// Alarm siren FB
FUNCTION_BLOCK FB_AlarmSiren IMPLEMENTS I_AlarmSiren
VAR
	sName				: STRING;				// Siren name
	nID					: INT;					// Alarm component ID
	
	ibTamper			AT %I* : BOOL;			// Active low tamper input
	fbLight				: FB_DigitalOut;		// Siren light digital output FB
	fbSiren				: FB_DigitalOut;		// Siren sound digital output FB
	
	bTamper				: BOOL;					// True if the siren is tampered with
	
	bTamperTrigger		: BOOL;					// True when the tamper sensor is triggered (one cycle)
	
	stHMI				: ST_AlarmSirenHMI;		// HMI data
END_VAR

// Run this method every cycle
METHOD Execute
VAR_INST
	fbTamper	: R_TRIG;		// Tamper rising edge
END_VAR
// Convert active low inputs
bTamper := NOT ibTamper;

// Run FBs
fbTamper(CLK := bTamper);

// Check trigger
bTamperTrigger := fbTamper.Q;

// Update HMI
UpdateHMI();
END_METHOD

METHOD FB_init : BOOL
VAR_INPUT
	bInitRetains	: BOOL;		// if TRUE, the retain variables are initialized (warm start / cold start)
	bInCopyCode		: BOOL;		// if TRUE, the instance afterwards gets moved into the copy code (online change)
	
	sSirenName		: STRING;	// Siren name
	nSirenID		: INT;		// Sensor ID
END_VAR
sName := sSirenName;
nID := nSirenID;
END_METHOD

// Returns the HMI data
PROPERTY HmiData : ST_AlarmSirenHMI
GET
HmiData := stHMI;
END_GET
END_PROPERTY

// Get the alarm component ID of the siren
PROPERTY ID : INT
GET
ID := nID;
END_GET
END_PROPERTY

// Set siren light
METHOD SetLight
VAR_INPUT
	eCommand	: E_DOCommand;		// Siren digital output command
END_VAR
// Set siren digital output command
fbLight.SetCommand(eCommandIn := eCommand);
END_METHOD

// Set siren sound
METHOD SetSound
VAR_INPUT
	eCommand	: E_DOCommand;		// Siren sound digital output command
END_VAR
// Set the siren digital output command
fbSiren.SetCommand(eCommandIn := eCommand);
END_METHOD

// Returns true when the siren is tampered with (as long as the siren is tampered with)
PROPERTY Tamper : BOOL
GET
Tamper := bTamper;
END_GET
END_PROPERTY

// Returns true when the tamper sensor is triggered (one cycle)
PROPERTY TamperTrigger : BOOL
GET
TamperTrigger := bTamperTrigger;
END_GET
END_PROPERTY

// Update HMI
METHOD PRIVATE UpdateHMI
VAR
	stSirenHMI	: ST_HmiDigitalOut;
	stLightHMI	: ST_HmiDigitalOut;
END_VAR
// Get data
stSirenHMI := fbSiren.HmiData;
stLightHMI := fbLight.HmiData;

// Set HMI data
stHMI.sName := sName;
stHMI.nID := nID;
stHMI.bSiren := stSirenHMI.bValue;
stHMI.bLight := stLightHMI.bValue;
stHMI.bTamper := bTamper;
END_METHOD

END_FUNCTION_BLOCK

(* stored: Version 1.1.0.1, ProductVersion 3.1.4024.12
   POU FB_AlarmSiren: Id {bb17f071-7286-41d1-bc99-46b7a45f36c9}, SpecialFunc None
   Folder Methods: Id {5e628541-4344-477b-a281-0b3fc142337b}
   Folder Properties: Id {1d8db5bb-13a1-4335-976d-c1ff1ce48bd0}
   Method Execute: Id {70dc7394-9df3-494a-875d-52b5fd2c9299}
   Method FB_init: Id {9acdc407-6a6c-4961-92b3-f2af5e52d2d4}
   Property HmiData: Id {06ad8ee2-5edc-4ca1-8bdd-00cc4c074abb}
   Get Get: Id {a33e8f75-5063-4901-9b85-6e748ef24f6d}
   Property ID: Id {3f061ba0-6334-4174-800b-553072ea0b2d}
   Get Get: Id {b338a67c-185e-4200-a022-6d18a52d9cda}
   Method SetLight: Id {cd843fc6-ca1b-496c-a1d3-fe4d993b99c3}
   Method SetSound: Id {2333adb4-937b-4551-8298-ff05a5541996}
   Property Tamper: Id {90d49093-fed7-4a0b-bc91-27c754668288}
   Get Get: Id {4b69639c-26c8-4868-b58b-5b0f44875f7b}
   Property TamperTrigger: Id {5c0c88fa-1b21-427a-aec3-222a246b0bf9}
   Get Get: Id {79a68602-190c-4328-ba89-7d471aad2891}
   Method UpdateHMI: Id {2be49e35-556a-4755-9e72-9f1b366da3a3} *)
